TYPE PLCOpenCommandInternal :
STRUCT
	_Execute : BOOL;
	_Trig : BOOL;
	_status : PLCOpenStatusBase;
	_remote : IPLCOpenCall;
	_nullRemote : PLCOpenNullRemote;
	_commandGroups : ARRAY[0..19] OF IPLCOpenGroup;
	_parameterReader : CopyPV;
END_STRUCT
END_TYPE

(* stored: Version 1.1.0.1, ProductVersion 3.1.4024.12
   DUT PLCOpenCommandInternal: Id {2586c15f-1927-4933-a282-856f73a5f588} *)
